DATA_BLOCK "DB_Setting"
TITLE =%version: 0.07 % CN: 20
//History:
//This version  %created_by: nlhdl %
//              %date_created: maandag 7 december 2015 15:58:42 %
//              %release: VI_RAW/RA_Dev %
//
//Modification History:                                   By:    Date:     Rev:
//----------------------------------------------------  -------  --------  -----
//ra#9751: Add source files ECS-P to VI_RAW             nlHdL    14-12-15   0.07
//ra#9751: Add source files ECS-P to VI_RAW             nlHdL    07-12-15   0.07
//7324: ECS-P General from the RD to RA for platform    nlHdL    06-07-15   0.07
//20643: DB moved to NON RETAIN memory                  nlHdL    16-09-14   0.07
//15797: Keyword release added                          nlwwij   26-09-13   0.06
//CR8000 Remove example code                            nlple    28-11-11   0.05
//CR7631 Insert key word for code generator             nlple    06-10-11   0.04
//Fixed up incompatible siemens keywords                nlMRe    25-10-10   0.03
//Added  TRZ0001_01_00 example                          nlMvK    22-10-10   0.02
//Initial revision                                      nlMRe    22-07-10   0.01
//
FAMILY : General
VERSION : 0.0
NON_RETAIN


  STRUCT
   common : "UDT_Common_Setting";
   Insert : INT ;	//Insertion point for the S7 Code Generator
  END_STRUCT ;
BEGIN
END_DATA_BLOCK

